// TwinCAT 3 PLC project Untitled1
// ProgramVersion: 3.1.4022.3
// libraries:
//   Tc2_Standard, * (Beckhoff Automation GmbH)
//   Tc2_System, * (Beckhoff Automation GmbH)
//   Tc3_Module, * (Beckhoff Automation GmbH)
//   VisuDialogs, * (System)
// project tree:
//   DUTs/ SafeState.TcDUT
//   / GlobalTextList.TcGTLO, PlcTask.TcTTO, Visualisierungsmanager.TcVMO (not stored)
//   GVLs/ GVL.TcGVL, GVL_Persistent.TcGVL
//   POUs/ MAIN.TcPOU, EdgeDetector.TcPOU
//   VISUs/ Visualization.TcVIS
// real-time tasks:
//   TASK PlcTask: cycle T#10ms, priority 20, ADS port 350

CONFIGURATION Untitled1
    RESOURCE PLC ON TwinCAT3
        TASK PlcTask(INTERVAL := T#10ms, PRIORITY := 20);
        PROGRAM MAIN WITH PlcTask : MAIN;
    END_RESOURCE
END_CONFIGURATION

// ---- DUTs/SafeState.TcDUT
{attribute 'qualified_only'}
{attribute 'strict'}
TYPE SafeState :
(
	Init		:= 0,
	Close		:= 1,
	CeckDigit	:= 2,
	WrongCode	:= 3,
	Open		:= 4
	
);
END_TYPE

// ---- GVLs/GVL.TcGVL
{attribute 'qualified_only'}
VAR_GLOBAL



END_VAR

// ---- GVLs/GVL_Persistent.TcGVL
{attribute 'qualified_only'}
VAR_GLOBAL PERSISTENT
	testIncr :INT;
	testStr : SafeState;
	

END_VAR

// ---- POUs/MAIN.TcPOU
PROGRAM MAIN
VAR
 // Edge Detector
	inputValue: BOOL := FALSE;
myEDG_var  : EdgeDetector;
riesingEdge :BOOL;
fallingEdge :BOOL;
	
currentSafeState  : SafeState := 0;
	
END_VAR

CASE currentSafeState OF
	
0:


1:


2:


3:


4:

END_CASE

//Implement Edge Detector
myEDG_var();
myEDG_var.inputValue := inputValue;
// Outputs from Edge Detection
riesingEdge :=myEDG_var.riesingEdge;
fallingEdge :=myEDG_var.fallingEdge;

END_PROGRAM

// ---- POUs/EdgeDetector.TcPOU
FUNCTION_BLOCK EdgeDetector
VAR_INPUT
	inputValue : BOOL ;
END_VAR

VAR_OUTPUT
	riesingEdge :BOOL;
	fallingEdge :BOOL;
END_VAR
VAR
	safeStatus:BOOL;
END_VAR



IF safeStatus = FALSE AND inputValue = TRUE THEN
riesingEdge:= TRUE;
fallingEdge:= FALSE;
ELSIF safeStatus = TRUE AND inputValue = FALSE THEN
fallingEdge:= TRUE;
riesingEdge:= FALSE;
END_IF
safeStatus := inputValue;

END_FUNCTION_BLOCK

// ---- VISUs/Visualization.TcVIS
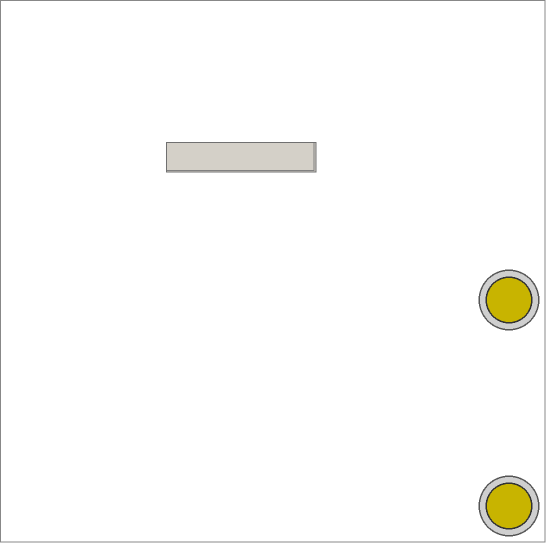
VISUALIZATION Visualization  // 546x543
    Button (166,142 150x30)
        OnMouseClick: toggle MAIN.inputValue
        OnMouseClick: toggle MAIN.inputValue
        OnMouseDown: write MAIN.inputValue via Default
    Lamp1 (474,265 70x70), variable: MAIN.riesingEdge, style: Lamp-Lamp1-Yellow
    Lamp1 (474,471 70x70), variable: MAIN.fallingEdge, style: Lamp-Lamp1-Yellow
END_VISUALIZATION
